Fanuc KAREL source: ka00121.KL

PROGRAM KA00121
%STACKSIZE=65535
%PRIORITY=65535
%NOLOCKGROUP
VAR
DST : INTEGER
-- UNRESOLVED DECLARATIONS (source type spelling not recovered)
-- SRC : ARRAY[2] OF TYPE_0x0018 (type_u16=0x2018)
BEGIN
SRC[1]=2
-- UNRESOLVED_PC line 8 opcodes [22 9D 33 B1 23] marker_code=19
END KA00121
